TYPE ST_LineDataOutCmd :
STRUCT
    Reserved : BOOL; // no command result
END_STRUCT
END_TYPE

(* stored: Version 1.1.0.1, ProductVersion 3.1.4024.12
   DUT ST_LineDataOutCmd: Id {de01f9ee-3120-4b39-95c5-cf56e519c203} *)
